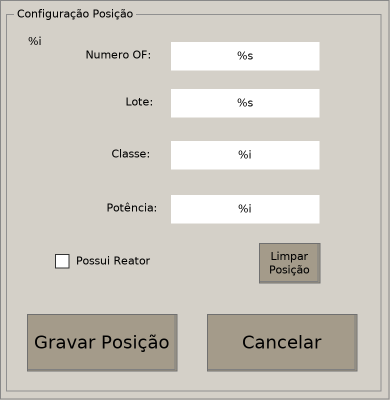
VISUALIZATION ConfigPosicao_3  // 390x400
VAR_IN_OUT
	bReator: BOOL;
	iOFnumber: INT;
	iSrlNumber: INT;
	
	
	
END_VAR
    GroupBox (6,6 375x385), "Configuração Posição"
        Checkbox (47,242 110x26), "Possui Reator", variable: gravarConfigPosicao021.bReator[2]
        Label (72,34 81x30), "Numero OF:"
        Textfield (164,35 150x30), "%s", text variable: GVL.cfgPos_OF021
            OnMouseDown: write the text variable via VisuDialogs.Numpad
        Label (97,133 56x30), "Classe:"
        Button (21,308 150x57), "Gravar Posição"
            OnMouseClick: CloseDialog Dialog=ConfigPosicao_3, Result=OK, NumpadKeypadSet=True
            OnMouseClick: execute { gravarConfigPosicao021(); }
        Button (201,308 150x57), "Cancelar"
            OnMouseClick: CloseDialog Dialog=ConfigPosicao_3, Result=Cancel, NumpadKeypadSet=True
        Button (253,237 61x40), "Limpar Posição"
            OnMouseClick: CloseDialog Dialog=ConfigPosicao_3, Result=Cancel, NumpadKeypadSet=True
            OnMouseClick: execute {
                gvl_p.aPositionsE021[gvl.actPos].numOF:='0';
                gvl_p.aPositionsE021[gvl.actPos].lote:='0';
                gvl_p.aPositionsE021[gvl.actPos].class:=0;
                gvl_p.aPositionsE021[gvl.actPos].pot:=0;
                gvl_p.aPositionsE021[gvl.actPos].cor:=0;
                IF gvl.totalPos[gvl.actEst] <> 0 THEN
                gvl.totalPos[gvl.actEst]:= gvl.totalPos[gvl.actEst] - 1;
                ELSE
                	gvl.totalPos[gvl.actEst] := 0;
                END_IF
                bReator:=false;
                ///// GERADOR DE LOG -------------------------------------------------------------
                gvl.envialog:= 'Posição Nº ';
                gvl.envialog:= concat(gvl.envialog, INT_TO_STRING(gvl.actPos));
                gvl.envialog:= concat(gvl.envialog,' foi limpa. ESTUFA 021');
                gvl.logRegister[gvl.actEst]:= gvl.envialog;
            }
        Textfield (164,134 150x30), "%i", text variable: GVL.cfgPos_Class021
            OnMouseDown: write the text variable via VisuDialogs.Numpad
        Textfield (164,188 150x30), "%i", text variable: GVL.cfgPos_Pot021
            OnMouseDown: write the text variable via VisuDialogs.Numpad
        Label (69,81 81x30), "Lote:"
    Label (104,193 56x30), "Potência:"
    Rectangle (24,30 22x23), "%i", text variable: GVL.actPos
    Textfield (170,88 150x30), "%s", text variable: GVL.cfgPos_LT021
        OnMouseDown: write the text variable via VisuDialogs.Keypad
END_VISUALIZATION

(* stored: Version 1.1.0.1, ProductVersion 3.1.4024.12
   Visu ConfigPosicao_3: Id {4db39272-76fd-4a7f-8493-da50291a50d7} *)
